Staubli VAL3: placetrial.pjx

--- placetrial.pjx ---
Parameters version=s7.6.2 stackSize=5000 millimeterUnit=true
Program file=start.pgx
Program file=stop.pgx
Data file=placetrial.dtx

--- placetrial.dtx ---
mdesc mNomSpeed
pointRx pick1 = {x=-473.86, y=319.07, z=-109, rx=180, ry=0, rz=-45, fatherId=world[0]}
pointRx pick1safe = {x=-473.86, y=319.07, z=-85, rx=-180, ry=0, rz=-45, fatherId=world[0]}
pointRx pick2 = {x=-473.860345, y=333.068871, z=-109, rx=179.999432, ry=0.000871, rz=-44.999837, fatherId=world[0]}
pointRx pick2safe = {x=-473.86, y=333.07, z=-85, rx=-180, ry=0, rz=-45, fatherId=world[0]}
pointRx pick3 = {x=-461.38, y=337.27, z=-109, rx=180, ry=0, rz=45, fatherId=world[0]}
pointRx pick3safe = {x=-461.38, y=337.27, z=-85, rx=-180, ry=0, rz=45, fatherId=world[0]}
pointRx place1 = {x=-494.006728, y=221.955751, z=-94, rx=179.999239, ry=0.000159, rz=-45.002417, fatherId=world[0]}
pointRx place1safe = {x=-494.005866, y=221.97, z=-85.004167, rx=179.99928, ry=0.000055, rz=-45.002417, fatherId=world[0]}
pointRx place2 = {x=-490.68, y=221.97, z=-94, rx=180, ry=0, rz=-45, fatherId=world[0]}
pointRx place2safe = {x=-490.68, y=221.97, z=-85, rx=-180, ry=0, rz=-45, fatherId=world[0]}
pointRx place3 = {x=-477.999337, y=204.167062, z=-94, rx=179.999117, ry=0.0011, rz=44.999832, fatherId=world[0]}
pointRx place3safe = {x=-477.999337, y=204.167062, z=-85, rx=179.999117, ry=0.0011, rz=44.999832, fatherId=world[0]}
